Staubli VAL3: readStrValue.pgx

public program readStrValue(num handle_, string x_sCellNumber, string& value_[], bool& result_[])
  local string strCell
begin
  // read contents of a cell
  // col_   : column of cell to read (column "A" -> 1, "B" -> 2, etc)
  // row_   : row of cell to read
  // value_ : contents of cell
  // result_: returns true if operation succeeded
  //          if false, check errorCode for error code of operation
  //
  nCommand[handle_]=coGV
  //call coord2Cell(col_,row_,strCell)
  //? "Command : gv"+x_sCellNumber
  call sendCommand(handle_,"gv"+x_sCellNumber,result_)
  if result_
    call readSocket(handle_,value_,result_)
  else
    value_=""
  endIf
end
